PROGRAM MAIN
VAR
END_VAR

END_PROGRAM

(* stored: Version 1.1.0.1
   POU MAIN: Id {3d574fcd-41b7-4104-9e93-8d967e83c80b} *)
